(* CODESYS project OSC_MQTT1.1.library
   Author: Peter Magnusson
   Title: MQTT Library
   Version: 1.0.0.1
   Description: Open Source CODESYS (OSC) MQTT Client library
   DefaultNamespace: OSC_MQTT
   Company: OSC

Project tree, tasks and I/O mapping:
  GenericDummyMasterDevice : Generic Master, WAGO Automation, order no. None, version 1.0.0.0
  libraries: CmpLog, 3.5.2.0 (System); Standard, 3.5.2.0 (System); CAA Types Extern, 3.5.3.0 (CAA Technical Workgroup); CmpErrors Interfaces, * (System); SysTypes Interfaces, * (System); IoStandard, 3.5.4.0 (System); SysMem, 3.5.4.0 (System); CAA Net Base Services, 3.5.4.0 (CAA Technical Workgroup); SysTarget, 3.5.4.0 (System); CmpEventMgr, 3.5.4.0 (System); CmpApp, 3.5.4.0 (System)
  MQTT/
    Function Blocks/
      function block MQTTClient [ST]: _writeByte, _connect, _write, _writeString, _writeWord, _disconnect, Publish, Subscribe, _Send, _Receive, _Keepalive
      function block MQTTPub [ST]
    Enums/
      data type CLIENTSTATE
      data type MESSAGETYPE
      data type QoS
    Structs/
      data type MQTTMESSAGE
    GlobalConstants/
      global variables Constants
*)

// MQTT/Enums/CLIENTSTATE
TYPE CLIENTSTATE :
(
	STOP:= 0,
	INIT,
	CONNECTING,
	CONNECTED,
	DISCONNECTING,
	DISCONNECTED,
	CLOSE,
	ERROR
);
END_TYPE

// MQTT/Enums/MESSAGETYPE
TYPE MESSAGETYPE :
(
	CONNECT 	:= 16#10,
	CONNACK 	:= 16#20,
	PUBLISH 	:= 16#30,
	PUBACK 		:= 16#40,
	SUBSCRIBE 	:= 16#80,
	SUBACK 		:= 16#90,
	UNSUBSCRIBE := 16#A0,
	UNSUBACK 	:= 16#B1,
	PINGREQ 	:= 16#C0,
	PINGRESP	:= 16#D0,
	DISCONNECT 	:= 16#E0
) BYTE;
END_TYPE

// MQTT/Enums/QoS
TYPE QoS :
(
	AtMostOnce:= 2#000,
	AtLeastOnce:= 2#010,
	ExactlyOnce:= 2#100
) BYTE;
END_TYPE

// MQTT/Structs/MQTTMESSAGE
TYPE MQTTMESSAGE :
STRUCT
	MessageType: MESSAGETYPE;
	DUP: BYTE;
	QoS: QoS;
	RetainMsg: BYTE;
	Length: BYTE;
	Payload: ARRAY[0..126] OF BYTE;
END_STRUCT
END_TYPE

// MQTT/GlobalConstants/Constants
{attribute 'qualified_only'}
VAR_GLOBAL CONSTANT	
	MQTTPROTOCOLVERSION : BYTE := BYTE#3;
	MQTT_MAX_PACKET_SIZE : BYTE := 128; //maximum packet size
	
	MQTT_MIN_KEEPALIVE : TIME := T#15S;	
	MQTT_DEFAULT_PORT : UINT := 1883;
	MQTT_MAX_CALLBACKS : INT :=3;
END_VAR

// MQTT/Function Blocks/MQTTClient
FUNCTION_BLOCK MQTTClient
VAR_INPUT
	sServerIP: STRING;
	uiPort: UINT := 1883;
	tKeepaliveInterval: TIME := T#15S;
	xEnable: BOOL;
END_VAR
VAR_OUTPUT
	xOnline: BOOL;
	dwError: DWORD;

END_VAR
VAR
	
	MQTT_TIMEAHEAD: TIME;
	Keepalive: TON;
	xKeepaliveEnabled: BOOL;
	xServerAlive:BOOL;

	TCPIPAddress: NBS.IP_ADDR;
	TCPClient: NBS.TCP_Client; /// FB TCP Client 
	TCPConnection: CAA.HANDLE; /// Handle to the established connection 
	TCPRead			: NBS.TCP_Read; (* FB TCP Read *)
	TCPWrite		: NBS.TCP_Write; (* FB TCP Writer *)
	RBUF: ARRAY[0..Constants.MQTT_MAX_PACKET_SIZE] OF BYTE; /// Receive Buffer
	SBUF: ARRAY[0..Constants.MQTT_MAX_PACKET_SIZE] OF BYTE; /// Send Buffer
	sLength: UINT;
	
	_nextMsgId: UINT;
	old_activate: BOOL := FALSE;
	eClientState: CLIENTSTATE;
	ePreviousClientState: CLIENTSTATE;
	cb: BYTE;
	idx1: INT;
	
	_isWriting: MESSAGETYPE; ///Command that is written.
	_hasMessage: BOOL; //has a received message to process
	msgIn: MQTTMESSAGE; //the last received message
	xSend: BOOL;
	
	
END_VAR


Keepalive(IN:=xKeepaliveEnabled, PT:= MQTT_TIMEAHEAD);
//first case of state
IF eClientState <> ePreviousClientState THEN
	CASE eClientState OF
		CLIENTSTATE.INIT:
			{IF defined (DEBUG_MQTTCLIENT)}
			LogAdd(STD_LOGGER,'MQTTClient',UDINT_TO_DINT(LogClass.LOG_INFO),0,0,'State.INIT');
			{END_IF}
			MQTT_TIMEAHEAD:= UDINT_TO_TIME(TIME_TO_UDINT(tKeepaliveInterval) / 3 * 2);// 2/3 to be paranoid 
		CLIENTSTATE.CONNECTING:
			{IF defined (DEBUG_MQTTCLIENT)}
			LogAdd(STD_LOGGER,'MQTTClient',UDINT_TO_DINT(LogClass.LOG_INFO),0,0,'State.CONNECTING');
			{END_IF}
		CLIENTSTATE.CONNECTED:
			{IF defined (DEBUG_MQTTCLIENT)}
			LogAdd(STD_LOGGER,'MQTTClient',UDINT_TO_DINT(LogClass.LOG_INFO),0,0,'State.CONNECTED');
			{END_IF}
		CLIENTSTATE.DISCONNECTING:
			{IF defined (DEBUG_MQTTCLIENT)}
			LogAdd(STD_LOGGER,'MQTTClient',UDINT_TO_DINT(LogClass.LOG_INFO),0,0,'State.DISCONNECTING');
			{END_IF}
		CLIENTSTATE.DISCONNECTED:
			{IF defined (DEBUG_MQTTCLIENT)}
			LogAdd(STD_LOGGER,'MQTTClient',UDINT_TO_DINT(LogClass.LOG_INFO),0,0,'State.DISCONNECTED');
			{END_IF}
		CLIENTSTATE.CLOSE:		
			{IF defined (DEBUG_MQTTCLIENT)}
			LogAdd(STD_LOGGER,'MQTTClient',UDINT_TO_DINT(LogClass.LOG_INFO),0,0,'State.CLOSE');
			{END_IF}
		CLIENTSTATE.ERROR:
			{IF defined (DEBUG_MQTTCLIENT)}
			LogAdd(STD_LOGGER,'MQTTClient',UDINT_TO_DINT(LogClass.LOG_INFO),0,0,'State.ERROR');
			{END_IF}
	END_CASE
END_IF
ePreviousClientState:= eClientState;

//every time the loop is in a certain state.
CASE eClientState OF
	
	CLIENTSTATE.STOP:
		xOnline := FALSE;
		
	CLIENTSTATE.INIT:
		SysMem.SysMemSet(ADR(SBUF), 0, SIZEOF(SBUF)); //clear send buffer;
		SysMem.SysMemSet(ADR(RBUF), 0, SIZEOF(RBUF)); //clear receive buffer;
		TCPIPAddress.sAddr := sServerIP;
		xSend:=FALSE;
		dwError := 0;
		sLength:=0;
		_hasMessage:= FALSE;
		_nextMsgId := 1;
		TCPWrite(xExecute:= FALSE);
		(* The client tries to establish a connection to a mqtt server *)
		TCPClient(xEnable:= TRUE, udiTimeOut:= 0, ipAddr:= TCPIPAddress, uiPort:= uiPort, hConnection=> TCPConnection);
		
			
		IF TCPClient.xActive THEN 
			eClientState:= CLIENTSTATE.CONNECTING;
			xServerAlive:=TRUE;
			THIS^._connect();
		ELSIF TCPClient.xError THEN
			
			eClientState:= CLIENTSTATE.ERROR;
		END_IF	
	(*------------------------- *)
	

	
	CLIENTSTATE.CONNECTED:
			xKeepaliveEnabled:= TRUE;
			xOnline:= TRUE;
	(*------------------------- *)
	
	CLIENTSTATE.DISCONNECTING:
			xKeepaliveEnabled:=FALSE;
			IF NOT xSend THEN
				eClientState:= DISCONNECTED;
			END_IF
	(*------------------------- *)	
	
	CLIENTSTATE.DISCONNECTED:		
		//logger('disconnected');
		xKeepaliveEnabled:=FALSE;
		eClientState:= CLOSE;
	(*------------------------- *)
	
	CLIENTSTATE.ERROR:
		xSend:=FALSE;
		TCPClient(xEnable := FALSE);
		eCLientState:= CLOSE;
		
	(*------------------------- *)
	
	CLIENTSTATE.CLOSE:		
		//logger('close');
		xServerAlive:=FALSE;
		xKeepaliveEnabled:=FALSE;
		old_activate := FALSE;
		xOnline:= FALSE;
		
		TCPWrite(xExecute:= FALSE);
		TCPRead(xEnable:=FALSE);
		TCPClient(xEnable:= FALSE);
		
		eClientState := CLIENTSTATE.STOP;
		
		
		
	(*------------------------- *)
	
END_CASE




//IPC1(IP:= DWORD#0, PORT:= WORD#0 , TIME_OUT:= TIMEOUT, IP_C:= IP_C1, S_BUF:= S_BUF1, R_BUF:= R_BUF1); (* MQTT Connection *)




IF NOT old_activate AND xEnable THEN
	eClientState := INIT;
	old_activate:= TRUE;
END_IF

IF NOT xEnable AND old_activate THEN
	{IF defined (DEBUG_MQTTCLIENT)}
	LogAdd(STD_LOGGER,'MQTTClient',UDINT_TO_DINT(LogClass.LOG_INFO),0,0,'Falling flank of xConnect ');
	{END_IF}
	THIS^._disconnect();
	old_activate:= FALSE;
END_IF

IF xSend AND TCPConnection = CAA.gc_hINVALID THEN
	xSend:= FALSE;
	IF eClientState <= CLIENTSTATE.DISCONNECTED THEN
		eClientState:= CLIENTSTATE.DISCONNECTED;
	END_IF
	
END_IF


IF TCPClient.xEnable AND TCPClient.xActive AND TCPClient.hConnection <> CAA.gc_hINVALID THEN
	THIS^._Keepalive();
	THIS^._Send();
	THIS^._Receive();
END_IF

METHOD PRIVATE _writeByte : INT
VAR_IN_OUT
	pos: UINT;
END_VAR
VAR_INPUT
	b: BYTE;
	pBuf: POINTER TO ARRAY[0..Constants.MQTT_MAX_PACKET_SIZE] OF BYTE;
END_VAR
//Add to current position according to size
pBuf^[pos]:= b;
//increase size
pos:= pos +1;
END_METHOD

METHOD PRIVATE _connect : BOOL
VAR_INPUT

END_VAR
VAR
	name: WSTRING:="01234567890123456789";
	dwId: DWORD;
	id: STRING;
	v: BYTE;
	w: UINT;
	length: UINT;
	MAX_NAME_LENGTH: UDINT := 20;
END_VAR

IF TCPClient.xActive THEN
		
	SysTarget.SysTargetGetNodeName(ADR(name), ADR(MAX_NAME_LENGTH));
	SysTarget.SysTargetGetId(ADR(dwId));
	id := CONCAT('mqttio/', WSTRING_TO_STRING(name));
	id := CONCAT(id, '-');
	id := CONCAT(id, DWORD_TO_STRING(dwId));
	
	 

	// {0x00,0x06,'M','Q','I','s','d','p',MQTTPROTOCOLVERSION};
	//leave room in the buffer for header and variable field length field
	length:=2;
	//start adding
	_writeByte(pos:=length, b:=16#0, pBuf := ADR(SBUF));
	_writeByte(pos:=length, b:=16#6, pBuf := ADR(SBUF));
	_writeString(pos:=length, msg:='MQIsdp');
	_writeByte(pos:=length, b:=Constants.MQTTPROTOCOLVERSION, pBuf := ADR(SBUF));
	
	//connect flags
	v := 16#2;//no will topic
	_writeByte(pos:=length, b:=v, pBuf := ADR(SBUF));
	
	//Keep Alive Timer
	_writeWord(pos:=length, w:= TIME_TO_WORD(tKeepaliveInterval/1000),  pBuf := ADR(SBUF)); 
	
	//client id length
	w:= INT_TO_UINT(LEN(id));
	_writeWord(pos:=length, w:=w,  pBuf := ADR(SBUF));
	//client id
	_writeString(pos:=length, msg:=id);
	_write(MESSAGETYPE.CONNECT, length);

END_IF
END_METHOD

METHOD PRIVATE _write : BOOL
VAR_INPUT
	header: MESSAGETYPE;
	length: UINT;
END_VAR
VAR
	len: BYTE;
END_VAR
IF TCPClient.xActive THEN	
	{IF defined (DEBUG_MQTTCLIENT)}
	LogAdd(STD_LOGGER,'MQTTClient',UDINT_TO_DINT(LogClass.LOG_INFO),0,0,CONCAT('Writing msg:', BYTE_TO_STRING(header) ));
	{END_IF}
	_isWriting:= header;
	len:= UINT_TO_BYTE(length);
	SBUF[0]:= header;
	IF len >= 2 THEN
		SBUF[1]:= len -2;
	ELSE
		SBUF[1]:= 0;
	END_IF
	
	IF(length<2) THEN
		length:= 2;
	END_IF
	sLength:= length;
	xSend:= TRUE;
END_IF
END_METHOD

METHOD PRIVATE _writeString
VAR_IN_OUT
	pos: UINT;
END_VAR
VAR_INPUT
	msg: STRING;
	
END_VAR

VAR
	ps : POINTER TO BYTE;
	end: UINT;
	i: UINT;
	length: UINT;
END_VAR
ps := ADR(msg);
length := INT_TO_UINT(LEN(msg));
end := MIN(pos + length, SIZEOF(SBUF));
IF end > 0 THEN end := end -1; END_IF;
FOR i := pos TO end DO
	SBUF[i] := ps^;
	ps := ps + 1;
END_FOR;
pos:=pos + length;
END_METHOD

METHOD PRIVATE _writeWord : INT
VAR_IN_OUT
	pos: UINT;
END_VAR
VAR_INPUT
	w: WORD;
	pBuf: POINTER TO ARRAY[0..Constants.MQTT_MAX_PACKET_SIZE] OF BYTE;
END_VAR
VAR
	v: BYTE;
	length: UINT;
END_VAR
length:= pos;
v:= UINT_TO_BYTE(SHR(w, 8));
_writeByte(pos:=length, b:=v, pBuf:=pBuf );
v:= UINT_TO_BYTE(w AND 16#FF);
_writeByte(pos:=length, b:=v, pBuf := pBuf); 
pos:= length;
END_METHOD

METHOD PRIVATE _disconnect
VAR_INPUT
END_VAR

VAR
	
END_VAR
{IF defined (DEBUG_MQTTCLIENT)}
LogAdd(STD_LOGGER,'MQTTClient',UDINT_TO_DINT(LogClass.LOG_INFO),0,0,'Calling _Disconnect');
{END_IF}
SysMem.SysMemSet(ADR(SBUF), 0, Constants.MQTT_MAX_PACKET_SIZE); //clear send buffer;
THIS^._write(MESSAGETYPE.DISCONNECT, 0);
eCLIENTSTATE:= CLIENTSTATE.DISCONNECTING;
END_METHOD

METHOD Publish
VAR_INPUT
	sTopic: STRING;
	sValue: STRING;
	xExecute: BOOL;
	bQos: BYTE;
	xRetain:BOOL;
END_VAR
VAR_OUTPUT
	xDone:BOOL;
END_VAR
VAR
	length: UINT;
	xBusyPublishing:BOOL; //will be set if publishing
	//EDITED FROM SR 19.08.2017 bBuf : ARRAY[0..Constants.MQTT_MAX_PACKET_SIZE] OF BYTE; /// Send Buffer
END_VAR

IF xExecute AND NOT xBusyPublishing THEN //Rising flank
	IF TCPClient.xActive THEN
		{IF defined (DEBUG_MQTTCLIENT)}
		LogAdd(STD_LOGGER,'MQTTClient',UDINT_TO_DINT(LogClass.LOG_INFO),0,0,'Publishing');
		{END_IF}
		xDone:=FALSE;
		xBusyPublishing:=TRUE;
		//sTopic := concat(sTopicPrefix, sTopic);
		length:= 2;//starting position in the buffer
		//EDITED FROM SR 19.08.2017_writeWord(pos:=length, w:= INT_TO_UINT(LEN(sTopic)), pBuf := ADR(bBuf));
		_writeWord(pos:=length, w:= INT_TO_UINT(LEN(sTopic)), pBuf := ADR(SBUF));
		_writeString(pos:=length, msg:=sTopic);
		IF bQos > 0 THEN //only send msg id if needed.
			_writeWord(pos:=length, w:= _nextMsgId, pBuf := ADR(SBUF));
		END_IF
		_writeString(pos:=length, msg:=sValue);
		_write(MESSAGETYPE.PUBLISH, length);
	END_IF
ELSIF NOT xExecute AND xBusyPublishing THEN //falling flank
	{IF defined (DEBUG_MQTTCLIENT)}
	LogAdd(STD_LOGGER,'MQTTClient',UDINT_TO_DINT(LogClass.LOG_INFO),0,0,'Publishing falling');
	{END_IF}
	xDone:=FALSE;
	xBusyPublishing:=FALSE;
ELSIF xExecute AND xBusyPublishing THEN //steady high
	//TODO:Wait for PUBACK if QoS >0
	IF NOT xSend THEN
		{IF defined (DEBUG_MQTTCLIENT)}
		LogAdd(STD_LOGGER,'MQTTClient',UDINT_TO_DINT(LogClass.LOG_INFO),0,0,'Publishing Done');
		{END_IF}
		xDone:=TRUE;
	END_IF
END_IF
END_METHOD

METHOD Subscribe : BOOL
VAR_INPUT
	sTopic: STRING;
	//pfbCallback: POINTER TO IMqttMessage;
END_VAR

VAR
	length: UINT;
END_VAR
//Save callback for later and send subscribe message
//m_Subscriptions.AddSub(sTopic:=sTopic, pfbCallback:=pfbCallback);

//leave room in the buffer for header and variable field length field
length:=2;

//topic and length of topic
_writeWord(pos:=length, INT_TO_UINT(LEN(sTopic)), pBuf := ADR(SBUF));
_writeString(pos:=length, msg:=sTopic);

//requested qos
_writeByte(pos:=length, b:=0, pBuf := ADR(SBUF));

_write(MESSAGETYPE.SUBSCRIBE, length);
END_METHOD

METHOD PRIVATE _Send
VAR_INPUT
END_VAR
IF xSend THEN
	

{IF defined (DEBUG_MQTTCLIENT)}
LogAdd(STD_LOGGER,'MQTTClient',UDINT_TO_DINT(LogClass.LOG_INFO),0,0,'Sending...');
{END_IF}
TCPWrite(xExecute:= TRUE, udiTimeOut:= 0, hConnection:= TCPConnection, szSize:= sLength, pData:= ADR(SBUF));
IF TCPWrite.xDone THEN 
	_nextMsgId:= _nextMsgId +1;				
	TCPWrite(xExecute:= FALSE);	
	xSend:= FALSE;
	sLength:= 0;		
	{IF defined (DEBUG_MQTTCLIENT)}
	LogAdd(STD_LOGGER,'MQTTClient',UDINT_TO_DINT(LogClass.LOG_INFO),0,0,'Sent');
	{END_IF}	
ELSIF TCPWrite.xError THEN
	//eCLIENTSTATE := CLIENTSTATE.ERROR;
	TCPWrite(xExecute:=FALSE);
	xSend:= FALSE;
	sLength:=0;
	{IF defined (DEBUG_MQTTCLIENT)}
	LogAdd(STD_LOGGER,'MQTTClient',UDINT_TO_DINT(LogClass.LOG_INFO),0,0,'Error Sending');
	{END_IF}
END_IF
IF _isWriting = MESSAGETYPE.DISCONNECT THEN
	eClientState := CLIENTSTATE.DISCONNECTED;
	xSend:=FALSE;
	{IF defined (DEBUG_MQTTCLIENT)}
	LogAdd(STD_LOGGER,'MQTTClient',UDINT_TO_DINT(LogClass.LOG_INFO),0,0,'Send Disconnect');
	{END_IF}
END_IF

END_IF
END_METHOD

METHOD PRIVATE _Receive
VAR_INPUT
END_VAR
TCPRead(xEnable:= TRUE, hConnection:= TCPConnection, szSize:= Constants.MQTT_MAX_PACKET_SIZE, pData:= ADR(RBUF));
IF TCPRead.xReady AND TCPRead.szCount > 0 THEN
	msgIn.MessageType := RBUF[0] AND 16#F0; //mask of first half
	msgIn.DUP := RBUF[0] AND 16#08;
	msgIn.QoS := RBUF[0] AND 16#06;
	msgIn.RetainMsg := RBUF[0] AND 1;
	msgIn.Length := RBUF[1]; //remaining length;
	SysMem.SysMemCpy(ADR(msgIn.Payload[0]), ADR(RBUF[2]), msgIn.Length);
	_hasMessage := TRUE;
	{IF defined (DEBUG_MQTTCLIENT)}
	LogAdd(STD_LOGGER,'MQTTClient',UDINT_TO_DINT(LogClass.LOG_INFO),0,0,CONCAT('Received:', BYTE_TO_STRING(msgIn.MessageType)));
	{END_IF}
ELSIF TCPRead.xError THEN
	eClientState := CLIENTSTATE.ERROR;
	{IF defined (DEBUG_MQTTCLIENT)}
	LogAdd(STD_LOGGER,'MQTTClient',UDINT_TO_DINT(LogClass.LOG_INFO),0,0,'Receive Error');
	{END_IF}
END_IF




IF _hasMessage THEN
//logger('hasMessage');	
	CASE _isWriting OF
		MESSAGETYPE.CONNECT:
			IF msgIn.MessageType = MESSAGETYPE.CONNACK THEN
				IF msgIn.Payload[1] = 0 THEN //connection accepted
					eClientState:= CONNECTED; 
					
				ELSE
					{IF defined (DEBUG_MQTTCLIENT)}
					LogAdd(STD_LOGGER,'MQTTClient',UDINT_TO_DINT(LogClass.LOG_INFO),0,0,'Could not authenticate');
					{END_IF}
					eClientState:= CLOSE;	
				END_IF
			END_IF
		(*----------------------------*)
		
		MESSAGETYPE.SUBSCRIBE:
			IF msgIn.MessageType = MESSAGETYPE.SUBACK THEN
				{IF defined (DEBUG_MQTTCLIENT)}
				LogAdd(STD_LOGGER,'MQTTClient',UDINT_TO_DINT(LogClass.LOG_INFO),0,0,'SUBACK');
				{END_IF}
			ELSE
				{IF defined (DEBUG_MQTTCLIENT)}
				LogAdd(STD_LOGGER,'MQTTClient',UDINT_TO_DINT(LogClass.LOG_INFO),0,0,'SUBACK EXPECTED BUT NOT RECEIVED');
				{END_IF}	
			END_IF
			
		(*----------------------------*)
		
		MESSAGETYPE.PINGREQ:
			IF msgIn.MessageType = MESSAGETYPE.PINGRESP THEN
				//server alive
				{IF defined (DEBUG_MQTTCLIENT)}
				LogAdd(STD_LOGGER,'MQTTClient',UDINT_TO_DINT(LogClass.LOG_INFO),0,0,'PINGRESP');
				{END_IF}
				xServerAlive:=TRUE;
			END_IF 
		(*----------------------------*)
		
	
	END_CASE
_hasMessage:= FALSE; //message is dealt with
END_IF
END_METHOD

METHOD PRIVATE _Keepalive
VAR_INPUT
END_VAR
//keepalive triggered
IF Keepalive.Q THEN
	xKeepaliveEnabled:= FALSE;
	IF NOT xServerAlive THEN
		//SOMETHING BAD HAPPENED
		{IF defined (DEBUG_MQTTCLIENT)}
		LogAdd(STD_LOGGER,'MQTTClient',UDINT_TO_DINT(LogClass.LOG_INFO),0,0,'Something bad happened with connection');
		{END_IF}
		eClientState:= CLOSE;
	ELSE
		//check if server is alive.
		xServerAlive:=FALSE;
		{IF defined (DEBUG_MQTTCLIENT)}
		LogAdd(STD_LOGGER,'MQTTClient',UDINT_TO_DINT(LogClass.LOG_INFO),0,0,'PINGREQ');
		{END_IF}
		_write(MESSAGETYPE.PINGREQ, 0);
	END_IF
END_IF
END_METHOD

END_FUNCTION_BLOCK

// MQTT/Function Blocks/MQTTPub
FUNCTION_BLOCK MQTTPub
VAR_INPUT
	pClient		:POINTER TO MQTTClient;
	sTopic		:STRING;
	sValue		:STRING;
	xExecute	:BOOL;
END_VAR
	
VAR_OUTPUT
	xDone		:BOOL;
END_VAR
VAR
	
END_VAR

IF xExecute THEN
	pClient^.Publish(sTopic:=sTopic, sValue:=sValue, bQos:=0, xRetain:=FALSE, xExecute:=TRUE, xDone => xDone);
END_IF

END_FUNCTION_BLOCK
